// TIA Portal project "Garden Sprinkler Control" (V17)
// Garden Sprinkler Control
// There is a garden sprinkler system with 4 zones. Zone 1 should operate for 15s, then Zone 2 should operate for 15s, then Zone 3 should operate for 15s and then Zone 4 should operate for 15s. The System will operate only if it is not raining and there is no one in the 4 zones.
// Note: The system will work even when there is someone in other zone

(* hardware
DEVICE "S7-1200 station_1"  S7-1200 Station
   slot 0: "Rack_0"  S7-1200 Rack  Rack  V1.0
   slot 1: "PLC_1"  CPU 1212C AC/DC/Rly  6ES7 212-1BE40-0XB0  V4.5
*)

// ===== PLC "PLC_1"  CPU 1212C AC/DC/Rly =====

VAR_GLOBAL   // PLC tag table "Default tag table"
   "Human_sensor_Zone_1" AT %I0.0 : Bool;
   "Human_sensor_Zone_2" AT %I0.1 : Bool;
   "Human_sensor_Zone_3" AT %I0.2 : Bool;
   "Human_sensor_Zone_4" AT %I0.3 : Bool;
   "Rain_Detection_Sensor" AT %I0.4 : Bool;
   "Switch_ON" AT %I0.5 : Bool;
   "Switch_OFF" AT %I0.6 : Bool;
   "Sprinkler_Zone_1" AT %Q0.0 : Bool;
   "Sprinkler_Zone_2" AT %Q0.1 : Bool;
   "Sprinkler_Zone_3" AT %Q0.2 : Bool;
   "Sprinkler_Zone_4" AT %Q0.3 : Bool;
   "Tag_1" AT %M0.0 : Bool;
   "Tag_2" AT %M0.1 : Bool;
   "Tag_3" AT %M0.2 : Bool;
   "Tag_4" AT %M0.3 : Bool;
   "Tag_5" AT %M0.4 : Bool;
   "Tag_6" AT %M0.5 : Bool;
END_VAR

// folder: System blocks/Program resources

DATA_BLOCK "IEC_Timer_0_DB"   // DB1
{ S7_Optimized_Access := 'TRUE' }
AUTHOR : Simatic
FAMILY : IEC
NAME : IEC_TMR
VERSION : 1.0
// stored: InstanceOfName IEC_TIMER
"IEC_TIMER"
BEGIN
END_DATA_BLOCK

DATA_BLOCK "IEC_Timer_0_DB_1"   // DB2
{ S7_Optimized_Access := 'TRUE' }
AUTHOR : Simatic
FAMILY : IEC
NAME : IEC_TMR
VERSION : 1.0
// stored: InstanceOfName IEC_TIMER
"IEC_TIMER"
BEGIN
END_DATA_BLOCK

DATA_BLOCK "IEC_Timer_0_DB_2"   // DB3
{ S7_Optimized_Access := 'TRUE' }
AUTHOR : Simatic
FAMILY : IEC
NAME : IEC_TMR
VERSION : 1.0
// stored: InstanceOfName IEC_TIMER
"IEC_TIMER"
BEGIN
END_DATA_BLOCK

DATA_BLOCK "IEC_Timer_0_DB_3"   // DB4
{ S7_Optimized_Access := 'TRUE' }
AUTHOR : Simatic
FAMILY : IEC
NAME : IEC_TMR
VERSION : 1.0
// stored: InstanceOfName IEC_TIMER
"IEC_TIMER"
BEGIN
END_DATA_BLOCK

DATA_BLOCK "IEC_Timer_0_DB_4"   // DB5
{ S7_Optimized_Access := 'TRUE' }
AUTHOR : Simatic
FAMILY : IEC
NAME : IEC_TMR
VERSION : 1.0
// stored: InstanceOfName IEC_TIMER
"IEC_TIMER"
BEGIN
END_DATA_BLOCK

DATA_BLOCK "IEC_Timer_0_DB_5"   // DB6
{ S7_Optimized_Access := 'TRUE' }
AUTHOR : Simatic
FAMILY : IEC
NAME : IEC_TMR
VERSION : 1.0
// stored: InstanceOfName IEC_TIMER
"IEC_TIMER"
BEGIN
END_DATA_BLOCK

DATA_BLOCK "IEC_Timer_0_DB_6"   // DB7
{ S7_Optimized_Access := 'TRUE' }
AUTHOR : Simatic
FAMILY : IEC
NAME : IEC_TMR
VERSION : 1.0
// stored: InstanceOfName IEC_TIMER
"IEC_TIMER"
BEGIN
END_DATA_BLOCK

DATA_BLOCK "IEC_Timer_0_DB_8"   // DB9
{ S7_Optimized_Access := 'TRUE' }
AUTHOR : Simatic
FAMILY : IEC
NAME : IEC_TMR
VERSION : 1.0
// stored: InstanceOfName IEC_TIMER
"IEC_TIMER"
BEGIN
END_DATA_BLOCK

DATA_BLOCK "IEC_Timer_0_DB_9"   // DB10
{ S7_Optimized_Access := 'TRUE' }
AUTHOR : Simatic
FAMILY : IEC
NAME : IEC_TMR
VERSION : 1.0
// stored: InstanceOfName IEC_TIMER
"IEC_TIMER"
BEGIN
END_DATA_BLOCK

// folder: (top level)

ORGANIZATION_BLOCK "Main"   // OB1, LAD, ProgramCycle
TITLE = "Main Program Sweep (Cycle)"
{ S7_Optimized_Access := 'TRUE' }
VERSION : 0.1
   VAR_INPUT
      Initial_Call : Bool;   // Initial call of this OB
      Remanence : Bool;   // =True, if remanent data are available
   END_VAR
   VAR_TEMP   // added for the SCL form of the ladder/FBD networks
      _w1 : Bool;
   END_VAR
BEGIN

REGION Network 1
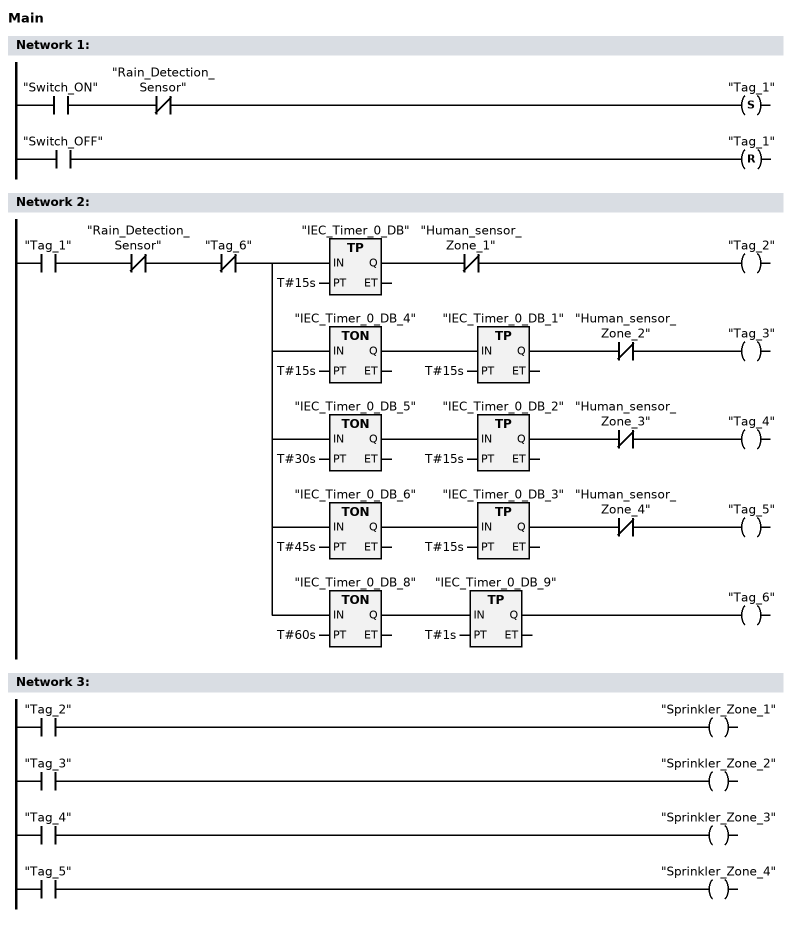
   RUNG wire#powerrail
      Contact( "Switch_ON" )
      I_Contact( "Rain_Detection_Sensor" )
      S_Coil( "Tag_1" )
   END_RUNG
   RUNG wire#powerrail
      Contact( "Switch_OFF" )
      R_Coil( "Tag_1" )
   END_RUNG
   // the same network as SCL:
   IF "Switch_ON" AND NOT "Rain_Detection_Sensor" THEN "Tag_1" := TRUE; END_IF;
   IF "Switch_OFF" THEN "Tag_1" := FALSE; END_IF;
END_REGION

REGION Network 2
   #_w1 := "Tag_1" AND NOT "Rain_Detection_Sensor" AND NOT "Tag_6";
   "IEC_Timer_0_DB".TP(IN := #_w1, PT := T#15s);
   "Tag_2" := "IEC_Timer_0_DB".Q AND NOT "Human_sensor_Zone_1";
   "IEC_Timer_0_DB_4".TON(IN := #_w1, PT := T#15s);
   "IEC_Timer_0_DB_1".TP(IN := "IEC_Timer_0_DB_4".Q, PT := T#15s);
   "Tag_3" := "IEC_Timer_0_DB_1".Q AND NOT "Human_sensor_Zone_2";
   "IEC_Timer_0_DB_5".TON(IN := #_w1, PT := T#30s);
   "IEC_Timer_0_DB_2".TP(IN := "IEC_Timer_0_DB_5".Q, PT := T#15s);
   "Tag_4" := "IEC_Timer_0_DB_2".Q AND NOT "Human_sensor_Zone_3";
   "IEC_Timer_0_DB_6".TON(IN := #_w1, PT := T#45s);
   "IEC_Timer_0_DB_3".TP(IN := "IEC_Timer_0_DB_6".Q, PT := T#15s);
   "Tag_5" := "IEC_Timer_0_DB_3".Q AND NOT "Human_sensor_Zone_4";
   "IEC_Timer_0_DB_8".TON(IN := #_w1, PT := T#60s);
   "IEC_Timer_0_DB_9".TP(IN := "IEC_Timer_0_DB_8".Q, PT := T#1s);
   "Tag_6" := "IEC_Timer_0_DB_9".Q;
END_REGION

REGION Network 3
   RUNG wire#powerrail
      Contact( "Tag_2" )
      Coil( "Sprinkler_Zone_1" )
   END_RUNG
   RUNG wire#powerrail
      Contact( "Tag_3" )
      Coil( "Sprinkler_Zone_2" )
   END_RUNG
   RUNG wire#powerrail
      Contact( "Tag_4" )
      Coil( "Sprinkler_Zone_3" )
   END_RUNG
   RUNG wire#powerrail
      Contact( "Tag_5" )
      Coil( "Sprinkler_Zone_4" )
   END_RUNG
   // the same network as SCL:
   "Sprinkler_Zone_1" := "Tag_2";
   "Sprinkler_Zone_2" := "Tag_3";
   "Sprinkler_Zone_3" := "Tag_4";
   "Sprinkler_Zone_4" := "Tag_5";
END_REGION
END_ORGANIZATION_BLOCK